(* PLC project Sin nombre, Desconocido Sin nombre 1 *)
(* stored: creationDateTime 2024-10-24T23:45:13, modificationDateTime 2024-10-25T01:01:30 *)

PROGRAM program0
  VAR
    sensor AT %IW0.0 : UINT := 0;
  END_VAR
  VAR CONSTANT
    min_baj : UINT := 33400;
    top_baj : UINT := 34500;
    top_alt : UINT := 36800;
  END_VAR
  VAR
    acum : UINT := 0;
    timer_norm : BOOL := 1;
    timer_alt : BOOL := 0;
    sal : BOOL;
    TON0 : TON;
    CTU_LINT0 : CTU_LINT;
    TON1 : TON;
    CTU_LINT1 : CTU_LINT;
  END_VAR
  VAR  (* added by the conversion: wires and edge detectors of the diagram *)
    _ADD30_ENO : BOOL;
    _ADD30_OUT : UINT;
    _DIV33_ENO : BOOL;
    _DIV33_OUT : UINT;
    _ADD36_ENO : BOOL;
    _ADD36_OUT : UINT;
    _DIV39_ENO : BOOL;
    _DIV39_OUT : UINT;
    R_TRIG1 : R_TRIG;
    R_TRIG2 : R_TRIG;
  END_VAR

(* LD diagram, written out as Structured Text *)
acum := (sensor + min_baj) / 2;
TON0(IN := TON0.Q OR timer_norm, PT := T#1s);
_ADD30_OUT := ADD(EN := TON0.Q, IN1 := sensor, IN2 := acum, ENO => _ADD30_ENO);
_DIV33_OUT := DIV(EN := _ADD30_ENO, IN1 := _ADD30_OUT, IN2 := 2, ENO => _DIV33_ENO);
IF _DIV33_ENO THEN acum := _DIV33_OUT; END_IF;
_ADD36_OUT := ADD(EN := timer_alt, IN1 := sensor, IN2 := acum, ENO => _ADD36_ENO);
_DIV39_OUT := DIV(EN := _ADD36_ENO, IN1 := _ADD36_OUT, IN2 := 2, ENO => _DIV39_ENO);
IF _DIV39_ENO THEN acum := _DIV39_OUT; END_IF;
TON1(IN := timer_alt, PT := T#1s);
timer_alt := TON1.Q;
R_TRIG1(CLK := timer_alt);
CTU_LINT1(CU := R_TRIG1.Q, PV := 1);
IF CTU_LINT1.Q THEN timer_norm := acum <= top_alt; END_IF;
R_TRIG2(CLK := TON0.Q);
CTU_LINT0(CU := R_TRIG2.Q, PV := 7);
IF CTU_LINT0.Q THEN GE(IN1 := acum, IN2 := top_baj); END_IF;
END_PROGRAM

CONFIGURATION Config0
  RESOURCE Res0 ON PLC
    TASK task0(INTERVAL := T#20ms, PRIORITY := 0);
    PROGRAM instance0 WITH task0 : program0;
  END_RESOURCE
END_CONFIGURATION
